Universal Robots PolyScope program: changePortTest.urp

Program changePortTest (installation=default directory=/home/ur/ursim/ursim-5.11.0.108249/programs createdIn=5.11.0.108249 lastSavedIn=5.11.0.108249 robotSerialNumber=20205501142)
Calibrated DH parameters: a=[0, -0.425, -0.3922, 0, 0, 0]; d=[0.1625, 0, 0, 0.1333, 0.0997, 0.0996]; alpha=[1.570796, 0, 0, 1.570796, -1.570796, 0]; deltaTheta=[0, 0, 0, 0, 0, 0]
BeforeStart
  Script: DP_rpc_swing = rpc_factory("xmlrpc","http://127.0.0.1:50012")
  port_ID := 0
Robot Program (runOnlyOnce=false)
  Script: port_ID = DP_rpc_swing.readPort()
  Halt
